% RSLogix 500 project Intro to PLC Job HO4 Connor Bolk.RSS, saved by version 10.00.00.00 %
PROJECT "UNTITLED"    % processor: Bul.1763 MicroLogix 1100 Series B %

PROGRAM FILES
  LAD 2   9 rungs

DATA FILES
  O0 OUTPUT  4 elements
  I1 INPUT  6 elements
  S2 STATUS  66 elements
  B3 BINARY  1 elements
  T4 TIMER  1 elements
  C5 COUNTER  1 elements
  R6 CONTROL  1 elements
  N7 INTEGER  1 elements
  F8 FLOAT  1 elements

LADDER 2
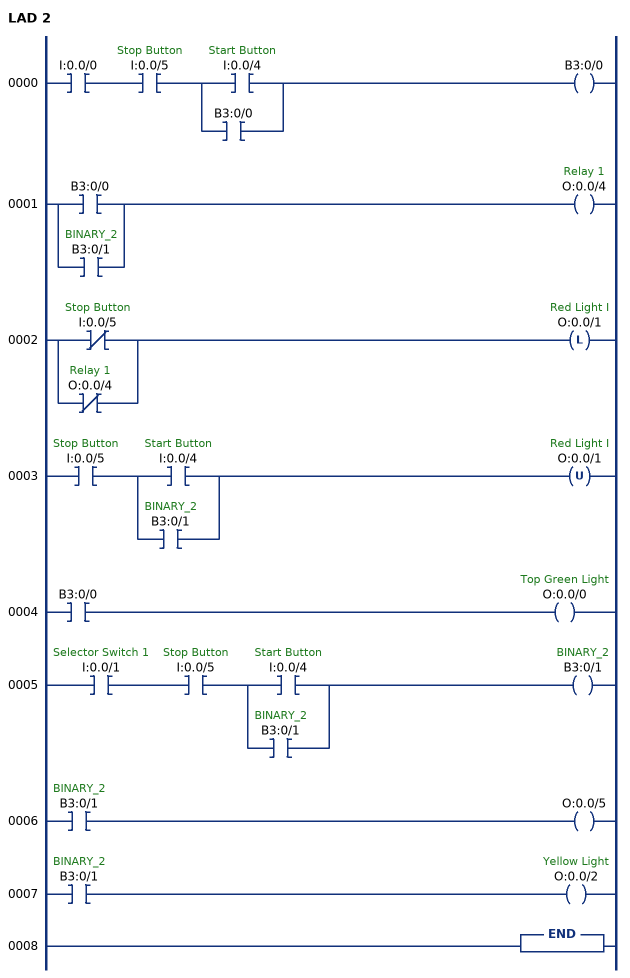
% Rung: 0 %
SOR XIC I:0.0/0 XIC I:0.0/5 BST XIC I:0.0/4 NXB XIC B3:0/0 BND OTE B3:0/0 EOR
%   XIC I:0.0/0  "Selector Switch 1" %
%   I:0.0/5  "Stop Button" %
%   XIC I:0.0/5  "Stop Button" %
%   I:0.0/4  "Start Button" %
%   XIC B3:0/0  "Binary 1" %
%   OTE B3:0/0  "Binary 1" %
% Rung: 1 %
SOR BST XIC B3:0/0 NXB XIC B3:0/1 BND OTE O:0.0/4 EOR
%   XIC B3:0/0  "Binary 1" %
%   B3:0/1  BINARY_2 %
%   O:0.0/4  "Relay 1" %
% Rung: 2 %
SOR BST XIO I:0.0/5 NXB XIO O:0.0/4 BND OTL O:0.0/1 EOR
%   I:0.0/5  "Stop Button" %
%   O:0.0/4  "Relay 1" %
%   O:0.0/1  I  "Red Light" %
% Rung: 3 %
SOR XIC I:0.0/5 BST XIC I:0.0/4 NXB XIC B3:0/1 BND OTU O:0.0/1 EOR
%   I:0.0/5  "Stop Button" %
%   XIC I:0.0/5  "Stop Button" %
%   I:0.0/4  "Start Button" %
%   B3:0/1  BINARY_2 %
%   O:0.0/1  I  "Red Light" %
% Rung: 4 %
SOR XIC B3:0/0 OTE O:0.0/0 EOR
%   XIC B3:0/0  "Binary 1" %
%   O:0.0/0  "Top Green Light" %
% Rung: 5 %
SOR XIC I:0.0/1 XIC I:0.0/5 BST XIC I:0.0/4 NXB XIC B3:0/1 BND OTE B3:0/1 EOR
%   I:0.0/1  "Selector Switch 1" %
%   I:0.0/5  "Stop Button" %
%   XIC I:0.0/5  "Stop Button" %
%   I:0.0/4  "Start Button" %
%   B3:0/1  BINARY_2 %
% Rung: 6 %
SOR XIC B3:0/1 OTE O:0.0/5 EOR
%   B3:0/1  BINARY_2 %
%   OTE O:0.0/5  "Relay 2" %
% Rung: 7 %
SOR XIC B3:0/1 OTE O:0.0/2 EOR
%   B3:0/1  BINARY_2 %
%   O:0.0/2  "Yellow Light" %
% Rung: 8 %
SOR END EOR

OTHER DOCUMENTED ADDRESSES
  B3:0/4  "BInary 4"
  O:0.0/3  "Green Light"
  O:1.0/1  "Red Light"
